(* PLC project  *)

PROGRAM BlocksXml
  VAR
    A : INT;
    B : INT;
    C : INT;
    D : INT;
    E : INT;
  END_VAR
  VAR  (* added by the conversion: wires and edge detectors of the diagram *)
    _ADD4_OUT : INT;
  END_VAR

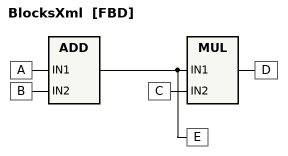
(* FBD diagram, written out as Structured Text *)
_ADD4_OUT := A + B;
D := _ADD4_OUT * C;
E := _ADD4_OUT;
END_PROGRAM
